FUNCTION FUN_PackBoolArrayToByte 	:BYTE
VAR_INPUT
		 Input						:ARRAY[0..7]OF BOOL;
END_VAR
VAR
		 idx						:INT;
END_VAR
//-----------------------------------------------oldschoo1

FUN_PackBoolArrayToByte := 0;

FOR idx:= 0 TO 7 
DO 
FUN_PackBoolArrayToByte := FUN_PackBoolArrayToByte OR TO_BYTE(SHL(BOOL_TO_INT(Input[idx]), idx)); 
END_FOR
//--------------------------------------------------------------------------------------oldschoo1

END_FUNCTION

(* stored: Version 1.1.0.1, ProductVersion 3.1.4024.12
   POU FUN_PackBoolArrayToByte: Id {b4b70a0d-48ed-44f1-9e25-9db0e8e7e3f3}, SpecialFunc None *)
